TYPE typeDataAxis :
STRUCT
	grabTime: ARRAY[1..20000] OF ULINT;
	grabData: ARRAY[1..20000] OF REAL;
	
END_STRUCT
END_TYPE

(* stored: Version 1.1.0.1, ProductVersion 3.1.4024.11
   DUT typeDataAxis: Id {a5f0e6ca-58f8-0739-2fd1-554532ca8cc4} *)
